// TIA Portal V20 export
TYPE "HMI_VlvL"
   STRUCT
      OpenMan : Bool;   // 1=Open: Open Command in Manual Mode
      CloseMan : Bool;   // 1=Close: Close Command in Manual Mode
      AutModOp : Bool;   // 1=Auto mode: auto mode by operator
      ManModOp : Bool := TRUE;   // 1=Manual mode: manual mode by operator
      LocalLi : Bool;   // 1=Local Mode: Local operation by field signal
      LocalOp : Bool;   // 1=Local Mode: Local operation by operator
      OosOp : Bool;   // 1=Oos mode: Oos mode by operator
      OpenLocal : Bool;   // 1=Open Local:Field Open Signal
      CloseLocal : Bool;   // 1=Close Local: Field Close Signal
      Monitor : Bool := TRUE;   // 1=Monitor ON, 0=Monitor OFF: Feedback monitor
      MonTiStatic : Real := 3.0;   // Monitoring time for unexpected change in any feedback [s]
      MonTiDynamic : Real := 3.0;   // Monitoring time for expected change of feedback [s]
      RstOp : Bool;   // Operator reset signal
      Permit_ST : Byte := BYTE#16#FF;   // Permit Signal Status
      Intlock_ST : Byte := BYTE#16#FF;   // Intlock Signal Status
      Protect_ST : Byte := BYTE#16#FF;   // Protect Signal Status
      CurrMon { ExternalWritable := 'False'} : DInt;   // Remaining monitoring time [s]
      Ctrl { ExternalWritable := 'False'} : Bool;   // Control output (dependent from SafePos)
      OS_PermOut { ExternalWritable := 'False'} : DWord := DWORD#16#FFFF_FFFF;   // Operator permission: output for OS
      OS_PermLog { ExternalWritable := 'False'} : DWord := DWORD#16#FFFF_FFFF;   // Operator permission: output for OS
      OpSt_Out { ExternalWritable := 'False'} : DWord;   // Enabled operator stations
      ST_Worst { ExternalWritable := 'False'} : Byte := 16#80;   // Worst signal status
      AutoST { ExternalWritable := 'False'} : Byte := 16#80;   // Worst Signal Status of the automatic commands
      Status1 { ExternalWritable := 'False'} : DWord;   // Status1 word
      Status2 { ExternalWritable := 'False'} : DWord;   // Status2 word
      Status3 { ExternalWritable := 'False'} : DWord;   // Status3 word
      Status4 { ExternalWritable := 'False'} : DWord;   // Status4 word
      AlarmState { ExternalWritable := 'False'} : Word;   // Alarm State for group display / Alarm Status for group display
   END_STRUCT;
END_TYPE
